Staubli VAL3: production.pgx

program production()
begin
  if taskStatus("txtLoad")!=-1
    taskKill("txtLoad")
    wait(taskStatus("txtLoad")==-1)
  endIf
  if taskStatus("motion")!=-1
    taskKill("motion")
    wait(taskStatus("motion")==-1)
  endIf
  //2015.06.23
  //taskCreateSync "txtLoad",0.004,bTxtLoad,read:fileRead(sTxtSelected)
  taskCreate "txtLoad",100,read:fileRead(sTxtSelected)
  taskCreate "motion",98,read:trajGrind()
  if taskStatus("prdMassage")==-1
    taskCreate "prdMassage",80,prdMassage()
  endIf
end
